FUNCTION_BLOCK Test_HandlerIsAddedToEventHandlerList EXTENDS TUnitTestBase
VAR
    TestEvent : TTestEvent;
    TestEventHandler : TTestEventHandler;
END_VAR

METHOD  Execute
TestEvent
    .ClearEventHandlers()
    .AddEventHandler(TestEventHandler);
    
Assertion.AssertEquals_UDINT(
    Expected      := 1,
    Actual        := TestEvent.EventHandlers.Count,
    ObjectName := _TestName,
    VariableName  := 'TestEvent.EventHandlers.Count');
    

_TestFinished := TRUE;
END_METHOD

END_FUNCTION_BLOCK

(* stored: Version 1.1.0.1, ProductVersion 3.1.4024.3
   POU Test_HandlerIsAddedToEventHandlerList: Id {de5a509b-4447-4128-ad4d-78293717de59}, SpecialFunc None
   Method Execute: Id {0847b3c0-8b97-40f0-8190-4dde8576ae1c} *)
